RoboDK station: project.rdk

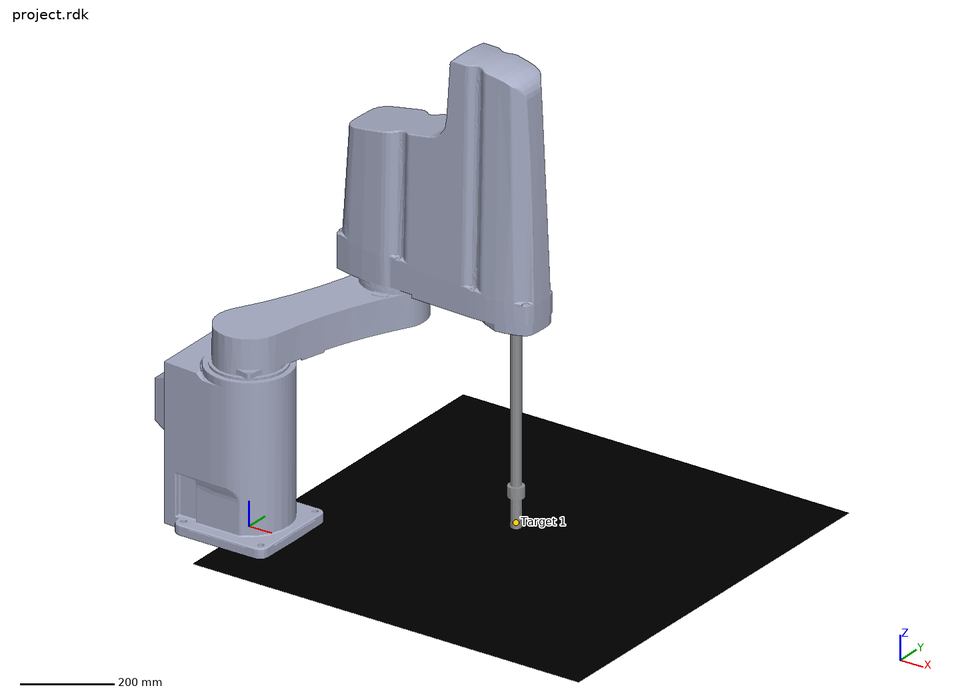
[picture v0: the station drawn from its stored meshes, robots at their saved joint values, targets as dots, program paths as lines]
Station project (saved by RoboDK 5.4.0). Poses are relative to the parent item; angles as X-Y-Z fixed-axis rotations.
  - Python program Prog1 (listed below)
  - frame Mitsubishi RH-12FH7035 Base at (-394.52, 0, 0) mm
    - robot Mitsubishi RH-12FH7035: 4 axes, payload 12 kg, reach 600 mm, repeatability 0.025 mm
        modified DH rows (alpha deg, a mm, theta deg, d mm): 0, 0, 0, 0; 0, 375, 0, 0; 0, 325, 0, 0 linear; 180, 0, 0, 0
        joint limits [-132, -150, 0, -360] to [132, 150, 300, 360]; home [0, 0, 350, 0]; saved at [69.772, -71.939, 0, 2.167]
    - target Target 1 (Cartesian target) at (454.42, 339.59, 0) mm; joints [130.825, -126.489, 0, -4.336] of Mitsubishi RH-12FH7035
  - object Plane 1m x 1m at (100, 300, -10) mm, size 1000 x 1000 x 0.5 mm, geometry from plane.sld
  - program Banawair1 last (0 instructions, listed below)
  - program 10 (0 instructions, listed below)
  - program mm2 (0 instructions, listed below)
  - program 10 (0 instructions, listed below)
  - program Banawair1 last (0 instructions, listed below)
  - program Banawair1 last (0 instructions, listed below)

--- Python program Prog1 ---
# Type help("robolink") or help("robodk") for more information
# Press F5 to run the script
# Documentation: https://robodk.com/doc/en/RoboDK-API.html
# Reference:     https://robodk.com/doc/en/PythonAPI/index.html
# Note: It is not required to keep a copy of this file, your python script is saved with the station

from robolink import *
from robodk import *

path = getOpenFile(r"Desktop") # open a window on at desktop to pick the csv file
data = LoadList(path) #Loading the (x,y,z) list
RDK = Robolink() # referring to the robot
robot = RDK.Item('', ITEM_TYPE_ROBOT) #apply the program on the picked robot.
target = RDK.Item('Target 1') #reference
position = target.Pose()
program_name = getFileName(path)
program = RDK.AddProgram(program_name, robot)
RDK.Render(False) # Turn off rendering (faster)

for i in range(len(data)):
    pi = position
    pi.setPos(data[i])
    target.setPose(pi)
    if i == 0:
        robot.MoveJ(target)
    else:

        robot.MoveL(target)

--- program Banawair1 last ---

--- program 10 ---

--- program mm2 ---

--- program 10 ---

--- program Banawair1 last ---

--- program Banawair1 last ---
